(*
Represents a receiver in the Broadcast system. Implements the necessary methods for receiving events and pairing signals.
Can be casted to `I_Component`.
*)
INTERFACE I_Receiver EXTENDS I_ReceiverNode, I_Tagged

END_INTERFACE

(* stored: Version 1.1.0.1
   Itf I_Receiver: Id {26bebb84-dbdb-4b7c-84a5-919778575944} *)
